Universal Robots PolyScope program: comb_fine_run.urp

Program comb_fine_run (installation=default directory=/programs/usbdisk createdIn=5.12.4.1101661 lastSavedIn=5.12.4.1101661)
Robot Program (runOnlyOnce=true)
  Script file /programs/usbdisk/comb_fine.script
    | def draw_svg():
    |   draw_z = 0.074940
    |   # home
    |   movel(p[0.598550, -0.129200, 0.105150, 2.249000, -2.194000, 0.000000], a=0.8, v=0.25, r=0.0)
    |   # stroke 0 (form id 0): simpleline
    |   movel(p[0.756629, -0.217706, 0.118080, 2.230000, -2.212000, 0.000000], a=0.8, v=0.25, r=0.0)
    |   movep(p[0.756629, -0.217706, draw_z, 2.230000, -2.212000, 0.000000], a=0.5, v=0.02, r=0.015000)
    |   movep(p[0.756169, -0.016748, draw_z, 2.230000, -2.212000, 0.000000], a=0.5, v=0.02, r=0.000000)
    |   movel(p[0.756169, -0.016748, 0.118080, 2.230000, -2.212000, 0.000000], a=0.8, v=0.25, r=0.0)
    |   # stroke 1 (form id 1): simpleline
    |   movel(p[0.749616, -0.217820, 0.118080, 2.230000, -2.212000, 0.000000], a=0.8, v=0.25, r=0.0)
    |   movep(p[0.749616, -0.217820, draw_z, 2.230000, -2.212000, 0.000000], a=0.5, v=0.02, r=0.015000)
    |   movep(p[0.749155, -0.016862, draw_z, 2.230000, -2.212000, 0.000000], a=0.5, v=0.02, r=0.000000)
    |   movel(p[0.749155, -0.016862, 0.118080, 2.230000, -2.212000, 0.000000], a=0.8, v=0.25, r=0.0)
    |   # stroke 2 (form id 2): simpleline
    |   movel(p[0.742602, -0.217934, 0.118080, 2.230000, -2.212000, 0.000000], a=0.8, v=0.25, r=0.0)
    |   movep(p[0.742602, -0.217934, draw_z, 2.230000, -2.212000, 0.000000], a=0.5, v=0.02, r=0.015000)
    |   movep(p[0.742142, -0.016976, draw_z, 2.230000, -2.212000, 0.000000], a=0.5, v=0.02, r=0.000000)
    |   movel(p[0.742142, -0.016976, 0.118080, 2.230000, -2.212000, 0.000000], a=0.8, v=0.25, r=0.0)
    |   # stroke 3 (form id 3): simpleline
    |   movel(p[0.735589, -0.218048, 0.118080, 2.230000, -2.212000, 0.000000], a=0.8, v=0.25, r=0.0)
    |   movep(p[0.735589, -0.218048, draw_z, 2.230000, -2.212000, 0.000000], a=0.5, v=0.02, r=0.015000)
    |   movep(p[0.735129, -0.017090, draw_z, 2.230000, -2.212000, 0.000000], a=0.5, v=0.02, r=0.000000)
    |   movel(p[0.735129, -0.017090, 0.118080, 2.230000, -2.212000, 0.000000], a=0.8, v=0.25, r=0.0)
    |   # stroke 4 (form id 4): simpleline
    |   movel(p[0.678355, -0.218979, 0.118080, 2.230000, -2.212000, 0.000000], a=0.8, v=0.25, r=0.0)
    |   movep(p[0.678355, -0.218979, draw_z, 2.230000, -2.212000, 0.000000], a=0.5, v=0.02, r=0.015000)
    |   movep(p[0.677895, -0.018021, draw_z, 2.230000, -2.212000, 0.000000], a=0.5, v=0.02, r=0.000000)
    |   movel(p[0.677895, -0.018021, 0.118080, 2.230000, -2.212000, 0.000000], a=0.8, v=0.25, r=0.0)
    |   # stroke 5 (form id 5): simpleline
    |   movel(p[0.672344, -0.219077, 0.118080, 2.230000, -2.212000, 0.000000], a=0.8, v=0.25, r=0.0)
    |   movep(p[0.672344, -0.219077, draw_z, 2.230000, -2.212000, 0.000000], a=0.5, v=0.02, r=0.015000)
    |   movep(p[0.671883, -0.018119, draw_z, 2.230000, -2.212000, 0.000000], a=0.5, v=0.02, r=0.000000)
    |   movel(p[0.671883, -0.018119, 0.118080, 2.230000, -2.212000, 0.000000], a=0.8, v=0.25, r=0.0)
    |   # stroke 6 (form id 6): simpleline
    |   movel(p[0.666333, -0.219174, 0.118080, 2.230000, -2.212000, 0.000000], a=0.8, v=0.25, r=0.0)
    |   movep(p[0.666333, -0.219174, draw_z, 2.230000, -2.212000, 0.000000], a=0.5, v=0.02, r=0.015000)
    |   movep(p[0.665872, -0.018217, draw_z, 2.230000, -2.212000, 0.000000], a=0.5, v=0.02, r=0.000000)
    |   movel(p[0.665872, -0.018217, 0.118080, 2.230000, -2.212000, 0.000000], a=0.8, v=0.25, r=0.0)
    |   # stroke 7 (form id 7): simpleline
    |   movel(p[0.660321, -0.219272, 0.118080, 2.230000, -2.212000, 0.000000], a=0.8, v=0.25, r=0.0)
    |   movep(p[0.660321, -0.219272, draw_z, 2.230000, -2.212000, 0.000000], a=0.5, v=0.02, r=0.015000)
    |   movep(p[0.659861, -0.018315, draw_z, 2.230000, -2.212000, 0.000000], a=0.5, v=0.02, r=0.000000)
    |   movel(p[0.659861, -0.018315, 0.118080, 2.230000, -2.212000, 0.000000], a=0.8, v=0.25, r=0.0)
    |   # stroke 8 (form id 8): simpleline
    |   movel(p[0.603087, -0.220203, 0.118080, 2.230000, -2.212000, 0.000000], a=0.8, v=0.25, r=0.0)
    |   movep(p[0.603087, -0.220203, draw_z, 2.230000, -2.212000, 0.000000], a=0.5, v=0.02, r=0.015000)
    |   movep(p[0.602627, -0.019246, draw_z, 2.230000, -2.212000, 0.000000], a=0.5, v=0.02, r=0.000000)
    |   movel(p[0.602627, -0.019246, 0.118080, 2.230000, -2.212000, 0.000000], a=0.8, v=0.25, r=0.0)
    |   # stroke 9 (form id 9): simpleline
    |   movel(p[0.598078, -0.220285, 0.118080, 2.230000, -2.212000, 0.000000], a=0.8, v=0.25, r=0.0)
    |   movep(p[0.598078, -0.220285, draw_z, 2.230000, -2.212000, 0.000000], a=0.5, v=0.02, r=0.015000)
    |   movep(p[0.597617, -0.019327, draw_z, 2.230000, -2.212000, 0.000000], a=0.5, v=0.02, r=0.000000)
    |   movel(p[0.597617, -0.019327, 0.118080, 2.230000, -2.212000, 0.000000], a=0.8, v=0.25, r=0.0)
    |   # stroke 10 (form id 10): simpleline
    |   movel(p[0.593068, -0.220366, 0.118080, 2.230000, -2.212000, 0.000000], a=0.8, v=0.25, r=0.0)
    |   movep(p[0.593068, -0.220366, draw_z, 2.230000, -2.212000, 0.000000], a=0.5, v=0.02, r=0.015000)
    |   movep(p[0.592608, -0.019409, draw_z, 2.230000, -2.212000, 0.000000], a=0.5, v=0.02, r=0.000000)
    |   movel(p[0.592608, -0.019409, 0.118080, 2.230000, -2.212000, 0.000000], a=0.8, v=0.25, r=0.0)
    |   # stroke 11 (form id 11): simpleline
    |   movel(p[0.588059, -0.220448, 0.118080, 2.230000, -2.212000, 0.000000], a=0.8, v=0.25, r=0.0)
    |   movep(p[0.588059, -0.220448, draw_z, 2.230000, -2.212000, 0.000000], a=0.5, v=0.02, r=0.015000)
    |   movep(p[0.587598, -0.019490, draw_z, 2.230000, -2.212000, 0.000000], a=0.5, v=0.02, r=0.000000)
    |   movel(p[0.587598, -0.019490, 0.118080, 2.230000, -2.212000, 0.000000], a=0.8, v=0.25, r=0.0)
    |   # stroke 12 (form id 12): simpleline
    |   movel(p[0.530825, -0.221379, 0.118080, 2.230000, -2.212000, 0.000000], a=0.8, v=0.25, r=0.0)
    |   movep(p[0.530825, -0.221379, draw_z, 2.230000, -2.212000, 0.000000], a=0.5, v=0.02, r=0.015000)
    |   movep(p[0.530365, -0.020421, draw_z, 2.230000, -2.212000, 0.000000], a=0.5, v=0.02, r=0.000000)
    |   movel(p[0.530365, -0.020421, 0.118080, 2.230000, -2.212000, 0.000000], a=0.8, v=0.25, r=0.0)
    |   # stroke 13 (form id 13): simpleline
    |   movel(p[0.526818, -0.221444, 0.118080, 2.230000, -2.212000, 0.000000], a=0.8, v=0.25, r=0.0)
    |   movep(p[0.526818, -0.221444, draw_z, 2.230000, -2.212000, 0.000000], a=0.5, v=0.02, r=0.015000)
    |   movep(p[0.526357, -0.020486, draw_z, 2.230000, -2.212000, 0.000000], a=0.5, v=0.02, r=0.000000)
    |   movel(p[0.526357, -0.020486, 0.118080, 2.230000, -2.212000, 0.000000], a=0.8, v=0.25, r=0.0)
    |   # stroke 14 (form id 14): simpleline
    |   movel(p[0.522810, -0.221509, 0.118080, 2.230000, -2.212000, 0.000000], a=0.8, v=0.25, r=0.0)
    |   movep(p[0.522810, -0.221509, draw_z, 2.230000, -2.212000, 0.000000], a=0.5, v=0.02, r=0.015000)
    |   movep(p[0.522349, -0.020552, draw_z, 2.230000, -2.212000, 0.000000], a=0.5, v=0.02, r=0.000000)
    |   movel(p[0.522349, -0.020552, 0.118080, 2.230000, -2.212000, 0.000000], a=0.8, v=0.25, r=0.0)
    |   # stroke 15 (form id 15): simpleline
    |   movel(p[0.518802, -0.221574, 0.118080, 2.230000, -2.212000, 0.000000], a=0.8, v=0.25, r=0.0)
    |   movep(p[0.518802, -0.221574, draw_z, 2.230000, -2.212000, 0.000000], a=0.5, v=0.02, r=0.015000)
    |   movep(p[0.518342, -0.020617, draw_z, 2.230000, -2.212000, 0.000000], a=0.5, v=0.02, r=0.000000)
    |   movel(p[0.518342, -0.020617, 0.118080, 2.230000, -2.212000, 0.000000], a=0.8, v=0.25, r=0.0)
    |   # stroke 16 (form id 16): simpleline
    |   movel(p[0.461569, -0.222505, 0.118080, 2.230000, -2.212000, 0.000000], a=0.8, v=0.25, r=0.0)
    |   movep(p[0.461569, -0.222505, draw_z, 2.230000, -2.212000, 0.000000], a=0.5, v=0.02, r=0.015000)
    |   movep(p[0.461108, -0.021548, draw_z, 2.230000, -2.212000, 0.000000], a=0.5, v=0.02, r=0.000000)
    |   movel(p[0.461108, -0.021548, 0.118080, 2.230000, -2.212000, 0.000000], a=0.8, v=0.25, r=0.0)
    |   # stroke 17 (form id 17): simpleline
    |   movel(p[0.458563, -0.222554, 0.118080, 2.230000, -2.212000, 0.000000], a=0.8, v=0.25, r=0.0)
    |   movep(p[0.458563, -0.222554, draw_z, 2.230000, -2.212000, 0.000000], a=0.5, v=0.02, r=0.015000)
    |   movep(p[0.458102, -0.021597, draw_z, 2.230000, -2.212000, 0.000000], a=0.5, v=0.02, r=0.000000)
    |   movel(p[0.458102, -0.021597, 0.118080, 2.230000, -2.212000, 0.000000], a=0.8, v=0.25, r=0.0)
    |   # stroke 18 (form id 18): simpleline
    |   movel(p[0.455557, -0.222603, 0.118080, 2.230000, -2.212000, 0.000000], a=0.8, v=0.25, r=0.0)
    |   movep(p[0.455557, -0.222603, draw_z, 2.230000, -2.212000, 0.000000], a=0.5, v=0.02, r=0.015000)
    |   movep(p[0.455097, -0.021646, draw_z, 2.230000, -2.212000, 0.000000], a=0.5, v=0.02, r=0.000000)
    |   movel(p[0.455097, -0.021646, 0.118080, 2.230000, -2.212000, 0.000000], a=0.8, v=0.25, r=0.0)
    |   # stroke 19 (form id 19): simpleline
    |   movel(p[0.452551, -0.222652, 0.118080, 2.230000, -2.212000, 0.000000], a=0.8, v=0.25, r=0.0)
    |   movep(p[0.452551, -0.222652, draw_z, 2.230000, -2.212000, 0.000000], a=0.5, v=0.02, r=0.015000)
    |   movep(p[0.452091, -0.021694, draw_z, 2.230000, -2.212000, 0.000000], a=0.5, v=0.02, r=0.000000)
    |   movel(p[0.452091, -0.021694, 0.118080, 2.230000, -2.212000, 0.000000], a=0.8, v=0.25, r=0.0)
    |   # park
    |   movel(p[0.598550, -0.129200, 0.105150, 2.249000, -2.194000, 0.000000], a=0.8, v=0.25, r=0.0)
    | end
    | draw_svg()
